ABB RobotStudio station: P2_Main.rspag

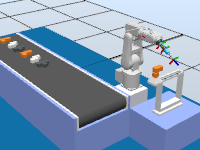
Station P2_Main (saved by RobotStudio 21.1.9385.0)
Layout (positions relative to the parent item):
  - IRB120_3_58__01 [mechanism, from Robots\IRB120_3_58_G_01.rslib] at (1547.5, 1227.5, 510) mm; joint values [0, 0, 0, 0, 0.5236, 0] (rad or m)
  - MyNewTool [mechanism] at (1911.85, 1227.5, 1104) mm, rotated rx 180 ry 60 rz 180 deg
      TCP MyNewTool at (0, 0, 0) mm, rotated rx 180 ry 0 rz 180 deg
      links: Čep
  - smc_gripper [mechanism, from P2\smc_gripper.rslib] at (1911.85, 1227.5, 1104) mm, rotated rx 180 ry 60 rz 180 deg
  - Conv_belt [part] at (-460, 1030, 390) mm, rotated rx 90 ry 0 rz 0 deg
  - Piece_L [part] at (-500, 715, 526.5) mm, rotated rx -90 ry 0 rz 0 deg
  - Piece_S [part] at (-250, 715, 526.5) mm, rotated rx -90 ry 0 rz 90 deg
  - Piece_T [part] at (-100, 765, 526.5) mm, rotated rx -90 ry 0 rz -90 deg
  - Piece_S_2 [part] at (350, 715, 526.5) mm, rotated rx -90 ry 0 rz 90 deg
  - Piece_L_2 [part] at (100, 715, 526.5) mm, rotated rx -90 ry 0 rz 0 deg
  - Piece_T_2 [part] at (500, 765, 526.5) mm, rotated rx -90 ry 0 rz -90 deg
  - Environment_3 [part]
  - Piece_Flip [part] at (1948.15, 1153.07, 875) mm, rotated rx 180 ry 0 rz 90 deg
  - Frame_1 [frame] at (0, 0, 60) mm
Attachment: MyNewTool is attached to IRB120_3_58__01 / Link6
Attachment: smc_gripper is attached to IRB120_3_58__01 / Link6
Targets, tools, work objects and paths stored in the station, written as RAPID:
! task (no controller)
MODULE CalibData
  PERS tooldata MyNewTool:=[TRUE,[[0,0,60],[1,0,0,0]],[0.3,[0,0,30.653],[1,0,0,0],0,0,0]];
  PERS tooldata smc_gripper:=[TRUE,[[0,0.004,197.001],[1,0,0,0]],[1,[0.207,-0.496,71.18],[1,0,0,0],0,0,0]];
ENDMODULE

